// TIA Portal V19 export
TYPE "C106_VAR_IF_MVI_TYPIC"
   STRUCT
      PWR1 { ExternalAccessible := 'False'; ExternalVisible := 'False'; ExternalWritable := 'False'} : Real;   // Geleverde actief vermogen per aggregaat
      PWR2 { ExternalAccessible := 'False'; ExternalVisible := 'False'; ExternalWritable := 'False'} : Real;   // Geleverde reactief vermogen per aggregaat
      SPA1 { ExternalAccessible := 'False'; ExternalVisible := 'False'; ExternalWritable := 'False'} : Real;   // Spanningsniveau lijn 1
      SPA2 { ExternalAccessible := 'False'; ExternalVisible := 'False'; ExternalWritable := 'False'} : Real;   // Spanningsniveau lijn 2
      SPA3 { ExternalAccessible := 'False'; ExternalVisible := 'False'; ExternalWritable := 'False'} : Real;   // Spanningsniveau lijn 3
      PSU_STO { ExternalAccessible := 'False'; ExternalVisible := 'False'; ExternalWritable := 'False'} : Bool;   // Storing door een fout op de UPS
      PSU_AUT { ExternalAccessible := 'False'; ExternalVisible := 'False'; ExternalWritable := 'False'} : Bool;   // Verzamelalarm actief: de beveiliging van de hulpvoeding is getript
      EXT_AUT { ExternalAccessible := 'False'; ExternalVisible := 'False'; ExternalWritable := 'False'} : Bool;   // Externe (hoofd) beveiliging aangesproken
      EXT_HW { ExternalAccessible := 'False'; ExternalVisible := 'False'; ExternalWritable := 'False'} : Bool;   // Sturings hardware (PLC) in storing
      STO { ExternalAccessible := 'False'; ExternalVisible := 'False'; ExternalWritable := 'False'} : Struct   // Opsomming van alle storingen
         A001 : Bool;   // Beveiliging aangesproken
         A002 : Bool;   // Hoogspanningsverdeelbord in storing
         A003 : Bool;   // Algemene storing hoogspanningsverdeelbord
         A004 : Bool;   // Alarm door een fout op de UPS
         A005 : Bool;   // Verzamelalarm actief: de beveiliging van de hulpvoeding is getript
      END_STRUCT;
   END_STRUCT;
END_TYPE
